// Interface for a Protocol Buffers message, supporting parsing from ST_ParserInternalState
// and writing to ST_WriterInternalState 
INTERFACE I_BufferMessage EXTENDS I_Message

METHOD InternalMergeFrom : HRESULT
VAR_IN_OUT
    fbCtx   : FB_ParseContext;
END_VAR
END_METHOD

METHOD InternalWriteTo : HRESULT
VAR_IN_OUT
    stState : ST_WriterInternalState;
END_VAR
END_METHOD

END_INTERFACE

(* stored: Version 1.1.0.1
   Itf I_BufferMessage: Id {f56f1e78-191a-4f3f-a73b-845a03427efc}
   Method InternalMergeFrom: Id {df371adf-7072-49a2-bfce-dcd90b23f2cc}
   Method InternalWriteTo: Id {4cb8226f-7662-47a8-94db-f4100d4b36d0} *)
